PROGRAM VisuInit
VAR_INPUT
	TFHandler : TextfieldInputHandler;
END_VAR

//VisuElems.g_VisuEventManager.SetEditBoxEventHandler(handler := TFHandler);

END_PROGRAM

(* stored: Version 1.1.0.1, ProductVersion 3.1.4024.12
   POU VisuInit: Id {f250eaae-ddf3-4905-b7d9-e7cd5944ef1b}, SpecialFunc None *)
